{attribute 'qualified_only'}
{attribute 'strict'}
TYPE E_LightgridType :
(
	WidthRight,
	WidthLeft,
	Height
);
END_TYPE

(* stored: Version 1.1.0.1, ProductVersion 3.1.4024.9
   DUT E_LightgridType: Id {67043294-7268-4d25-976b-a8d1976fdc51} *)
